PROGRAM MAIN
VAR
	// BOOLS for Errors and Machine condition created here
	bMachineOn: BOOL := TRUE;
	bEStopPressed: BOOL := FALSE;
	bMachineOverload: BOOL := FALSE;
	bDoorOpen: BOOL := FALSE;
	bMasterFault: BOOL := FALSE;
	bReset: BOOL := FALSE;
	bErrorPresent: BOOL := FALSE;
	
END_VAR

// IF statement detecting if any errors are currently active and activating memory if condition is met.
IF bEStopPressed OR bMachineOverload OR bDoorOpen THEN
	bMasterFault := TRUE;
	bErrorPresent:= TRUE;
ELSE;
	bErrorPresent := FALSE;
END_IF;

// Another If statement for activating reset, enabling only when no errors are present.
IF bReset AND NOT bErrorPresent THEN
	bMasterFault := FALSE;
END_IF;

//Master Fault Memory disabling machine if it is currently active and keeping the machine running otherwise.
IF bMasterFault THEN
	bMachineOn := FALSE;
ELSE;
	bMachineOn := TRUE;
END_IF;

END_PROGRAM

(* stored: Version 1.1.0.1, ProductVersion 3.1.4024.16
   POU MAIN: Id {81ce9aaf-6b63-44e6-9a46-06e3ba48373a}, SpecialFunc None *)
